FUNCTION_BLOCK Pulse
VAR_INPUT
	Pulse_time : TIME; // Az impulzus ideje, ennyi idő után kapcsol le
END_VAR
VAR_OUTPUT
	
END_VAR

VAR
clk :TON;

END_VAR
VAR_IN_OUT
	SIGNAL  : BOOL; // A jel amit kapcsolni kell
END_VAR

clk(IN:=SIGNAL,PT:=Pulse_time);

IF clk.Q THEN
	SIGNAL := FALSE;
		
END_IF

END_FUNCTION_BLOCK

(* stored: Version 1.1.0.1, ProductVersion 3.1.4024.11
   POU Pulse: Id {28473afe-7638-47f6-80ec-3b397164e5a1}, SpecialFunc None *)
